INTERFACE I_Table EXTENDS __System.IQueryInterface

PROPERTY INTERNAL _InternalTable : REFERENCE TO ST_NciFeedGroupTable
GET
END_GET
END_PROPERTY

METHOD AddAxisDynamics : BOOL
VAR_INPUT
	displayIndex : UDINT;
    axis : I_Axis;
    acceleration : LREAL(0.000001-99999999);
    deceleration : LREAL(0.000001-99999999);
    jerk: LREAL(0.000001-99999999);
END_VAR
END_METHOD

METHOD AddBaseFrame : BOOL
VAR_INPUT
    displayIndex : UDINT;
    shiftX : LREAL;
    shiftY : LREAL;
    shiftZ : LREAL;
    rotationX : LREAL;
    rotationY : LREAL;
    rotationZ : LREAL;
    shiftQ1 : LREAL;
    shiftQ2 : LREAL;
    shiftQ3 : LREAL;
    shiftQ4 : LREAL;
    shiftQ5 : LREAL;
END_VAR
END_METHOD

METHOD AddBaseFrame3D : BOOL
VAR_INPUT
    displayIndex : UDINT;
    shiftX : LREAL;
    shiftY : LREAL;
    shiftZ : LREAL;
    rotationX : LREAL;
    rotationY : LREAL;
    rotationZ : LREAL;
END_VAR
END_METHOD

METHOD AddBezier3rdOrder : BOOL
VAR_INPUT
	displayIndex : UDINT;
    controlPoint1X : LREAL;
    controlPoint1Y : LREAL;
    controlPoint1Z : LREAL;
    controlPoint2X : LREAL;
    controlPoint2Y : LREAL;
    controlPoint2Z : LREAL;
	endPositionX : LREAL;
	endPositionY : LREAL;
	endPositionZ : LREAL;
	endPositionQ1 : LREAL;
	endPositionQ2 : LREAL;
	endPositionQ3 : LREAL;
	endPositionQ4 : LREAL;
	endPositionQ5 : LREAL;
	velocity : LREAL(0.000001-99999999);
	accurateStop : BOOL; // velocity at end == 0
END_VAR
END_METHOD

METHOD AddBezier3rdOrder3D : BOOL
VAR_INPUT
	displayIndex : UDINT;
    controlPoint1X : LREAL;
    controlPoint1Y : LREAL;
    controlPoint1Z : LREAL;
    controlPoint2X : LREAL;
    controlPoint2Y : LREAL;
    controlPoint2Z : LREAL;
	endPositionX : LREAL;
	endPositionY : LREAL;
	endPositionZ : LREAL;
	velocity : LREAL(0.000001-99999999);
	accurateStop : BOOL; // velocity at end == 0
END_VAR
END_METHOD

METHOD AddBezier5thOrder : BOOL
VAR_INPUT
	displayIndex : UDINT;
    controlPoint1X : LREAL;
    controlPoint1Y : LREAL;
    controlPoint1Z : LREAL;
    controlPoint2X : LREAL;
    controlPoint2Y : LREAL;
    controlPoint2Z : LREAL;
    controlPoint3X : LREAL;
    controlPoint3Y : LREAL;
    controlPoint3Z : LREAL;
    controlPoint4X : LREAL;
    controlPoint4Y : LREAL;
    controlPoint4Z : LREAL;
	endPositionX : LREAL;
	endPositionY : LREAL;
	endPositionZ : LREAL;
	endPositionQ1 : LREAL;
	endPositionQ2 : LREAL;
	endPositionQ3 : LREAL;
	endPositionQ4 : LREAL;
	endPositionQ5 : LREAL;
	velocity : LREAL(0.000001-99999999);
	accurateStop : BOOL; // velocity at end == 0
END_VAR
END_METHOD

METHOD AddBezier5thOrder3D : BOOL
VAR_INPUT
	displayIndex : UDINT;
    controlPoint1X : LREAL;
    controlPoint1Y : LREAL;
    controlPoint1Z : LREAL;
    controlPoint2X : LREAL;
    controlPoint2Y : LREAL;
    controlPoint2Z : LREAL;
    controlPoint3X : LREAL;
    controlPoint3Y : LREAL;
    controlPoint3Z : LREAL;
    controlPoint4X : LREAL;
    controlPoint4Y : LREAL;
    controlPoint4Z : LREAL;
	endPositionX : LREAL;
	endPositionY : LREAL;
	endPositionZ : LREAL;
	velocity : LREAL(0.000001-99999999);
	accurateStop : BOOL; // velocity at end == 0
END_VAR
END_METHOD

METHOD AddCircleCIP : BOOL
VAR_INPUT
	displayIndex : UDINT;
	endPositionX : LREAL;
	endPositionY : LREAL;
	endPositionZ : LREAL;
	arcPointX : LREAL;
	arcPointY : LREAL;
	arcPointZ : LREAL;
	endPositionQ1 : LREAL;
	endPositionQ2 : LREAL;
	endPositionQ3 : LREAL;
	endPositionQ4 : LREAL;
	endPositionQ5 : LREAL;
	velocity : LREAL(0.000001-99999999);
	accurateStop : BOOL; // velocity at end == 0
END_VAR
END_METHOD

METHOD AddCircleCIP3D : BOOL
VAR_INPUT
	displayIndex : UDINT;
	endPositionX : LREAL;
	endPositionY : LREAL;
	endPositionZ : LREAL;
	arcPointX : LREAL;
	arcPointY : LREAL;
	arcPointZ : LREAL;
	velocity : LREAL(0.000001-99999999);
	accurateStop : BOOL; // velocity at end == 0
END_VAR
END_METHOD

METHOD AddCircleOnPlane : BOOL
VAR_INPUT
	displayIndex : UDINT;
	endPositionX : LREAL;
	endPositionY : LREAL;
	endPositionZ : LREAL;
	centerX : LREAL;
	centerY : LREAL;
	centerZ : LREAL;
	endPositionQ1 : LREAL;
	endPositionQ2 : LREAL;
	endPositionQ3 : LREAL;
	endPositionQ4 : LREAL;
	endPositionQ5 : LREAL;
	plane : StandardPlane := StandardPlane.XY;
	clockwise : BOOL;
	velocity : LREAL(0.000001-99999999);
	accurateStop : BOOL; // velocity at end == 0
END_VAR
END_METHOD

METHOD AddCircleOnPlane3D : BOOL
VAR_INPUT
	displayIndex : UDINT;
	endPositionX : LREAL;
	endPositionY : LREAL;
	endPositionZ : LREAL;
	centerX : LREAL;
	centerY : LREAL;
	centerZ : LREAL;
	plane : StandardPlane := StandardPlane.XY;
	clockwise : BOOL;
	velocity : LREAL(0.000001-99999999);
	accurateStop : BOOL; // velocity at end == 0
END_VAR
END_METHOD

METHOD AddDwellTime : BOOL
VAR_INPUT
	displayIndex : UDINT;
    dwellTime : LREAL(0.000001-99999999); // seconds
END_VAR
END_METHOD

METHOD AddFeedrateInterpolation : BOOL
VAR_INPUT
	displayIndex : UDINT;
	interpolationType : FeedrateInterpolation;
END_VAR
END_METHOD

METHOD AddLine : BOOL
VAR_INPUT
    displayIndex: UDINT;
    endPositionX: LREAL;
    endPositionY: LREAL;
    endPositionZ: LREAL;
    endPositionQ1: LREAL;
    endPositionQ2: LREAL;
    endPositionQ3: LREAL;
    endPositionQ4: LREAL;
    endPositionQ5: LREAL;
    velocity: LREAL(0.000001-99999999);
    rapidTraverse: BOOL;
    accurateStop: BOOL; // velocity at end == 0
END_VAR
END_METHOD

METHOD AddLine3D : BOOL
VAR_INPUT
    displayIndex: UDINT;
    endPositionX: LREAL;
    endPositionY: LREAL;
    endPositionZ: LREAL;
    velocity: LREAL(0.000001-99999999);
    rapidTraverse: BOOL;
    accurateStop: BOOL; // velocity at end == 0
END_VAR
END_METHOD

METHOD AddMFunctionWithHandshake : BOOL
VAR_INPUT
	displayIndex : UDINT;
    functionNumber : INT(0..159);
END_VAR
END_METHOD

METHOD AddPathDynamics : BOOL
VAR_INPUT
    displayIndex : UDINT;
    acceleration : LREAL(0.000001-99999999);
    deceleration : LREAL(0.000001-99999999);
    jerk : LREAL(0.000001-99999999);
END_VAR
END_METHOD

METHOD AddStart : BOOL
VAR_INPUT
	x : LREAL;
	y : LREAL;
	z : LREAL;
	q1 : LREAL;
	q2 : LREAL;
	q3 : LREAL;
	q4 : LREAL;
	q5 : LREAL;
END_VAR
END_METHOD

METHOD AddStart3D : BOOL
VAR_INPUT
	x : LREAL;
	y : LREAL;
	z : LREAL;
END_VAR
END_METHOD

METHOD DisableTangentialFollowing : BOOL
END_METHOD

METHOD DisableVertexSmoothing : BOOL
VAR_INPUT
	displayIndex : UDINT;
END_VAR
END_METHOD

METHOD EnableTangentialFollowing : BOOL
VAR_INPUT
    tangentialAxis : NciAxis; // axis used for tangential following
    pathAxis1 : NciAxis; // describing the plane e.g. x
    pathAxis2 : NciAxis; // e.g. y ==> g17, xy plane
    offset : LREAL; // geo tangent is 0 degree, counting is mathmatical positive
	criticalAngle : LREAL(0.000001-90);
    behaviour : TangentialFollowingBehaviour;
END_VAR
END_METHOD

METHOD EnableVertexSmoothing : BOOL
VAR_INPUT
	displayIndex : UDINT;
	blendType : VertexSmoothingBlendingType;
	subType : VertexSmoothingSubType; 
	radius : LREAL(0.000001-99999999);
END_VAR
END_METHOD

METHOD End : BOOL
END_METHOD

PROPERTY ErrorId : UDINT
GET
END_GET
END_PROPERTY

PROPERTY FilledRows : INT
GET
END_GET
END_PROPERTY

PROPERTY HasError : BOOL
GET
END_GET
END_PROPERTY

METHOD ResetAll : BOOL
END_METHOD

METHOD ResetTable : BOOL
END_METHOD

END_INTERFACE

(* stored: Version 1.1.0.1, ProductVersion 3.1.4024.12
   Itf I_Table: Id {739dd892-cb31-4bd0-a191-42ac4941c726}
   Property _InternalTable: Id {7b598730-f029-415a-b056-55b65e711f78}
   Get Get: Id {078af100-b2d1-44ec-a028-70c3bd4f11fe}
   Method AddAxisDynamics: Id {90b05305-7afb-4b84-85bb-ee24976dbbd8}
   Method AddBaseFrame: Id {afffafb0-7905-4a68-8a9d-9d617c15ab24}
   Method AddBaseFrame3D: Id {f4614335-b82a-47c3-9bee-2b6d18723083}
   Method AddBezier3rdOrder: Id {dac5ed2d-a91b-48eb-9950-3b9fb425d0a0}
   Method AddBezier3rdOrder3D: Id {4da67f00-46f0-416b-99fe-34dfe230497f}
   Method AddBezier5thOrder: Id {608ada7a-5786-4b63-adf2-4f2f4d22b371}
   Method AddBezier5thOrder3D: Id {5448bb54-6ec0-455c-b5b5-abe54411ded6}
   Method AddCircleCIP: Id {f044aea4-54b1-4049-a247-70896b69338f}
   Method AddCircleCIP3D: Id {326bb761-f8b9-428d-b787-7723655c4754}
   Method AddCircleOnPlane: Id {b4aaee45-5a64-4c78-bb6f-16a1f9e654e4}
   Method AddCircleOnPlane3D: Id {c9bf8cb5-0c5c-4f90-b503-fe16026c8d3f}
   Method AddDwellTime: Id {b6adeded-8b48-4167-8093-b8d002dcc967}
   Method AddFeedrateInterpolation: Id {5d6f284c-2f7d-4fbf-b57d-9c01ad6226bb}
   Method AddLine: Id {106e0278-8d7e-41d7-b6ef-895917ab3f3a}
   Method AddLine3D: Id {99855279-ecd0-41f0-99b1-2a5b21a9a526}
   Method AddMFunctionWithHandshake: Id {5f20215b-a091-4387-af2a-b5cdbe2e7b1b}
   Method AddPathDynamics: Id {3d54cbd2-cb38-43da-a49d-c93565722659}
   Method AddStart: Id {f3b32d87-ed5b-4ff7-ab74-18ab3d304a5b}
   Method AddStart3D: Id {1ee68d1d-485d-4f29-b4d1-78f0bd4ad3fa}
   Method DisableTangentialFollowing: Id {b0c3e73a-02de-4535-a428-d2afc05f3630}
   Method DisableVertexSmoothing: Id {e2c24514-b215-47a0-ab5e-791ad29a1996}
   Method EnableTangentialFollowing: Id {d1542920-828f-4dc4-bb27-e38798603e0a}
   Method EnableVertexSmoothing: Id {4a6ad671-c0c0-409a-bd30-08442afd78af}
   Method End: Id {83e2a824-c91c-4b2c-be28-ca32c6009d21}
   Property ErrorId: Id {88f45720-8df7-4ae7-a4d0-027d75f3ccab}
   Get Get: Id {d03d66d0-6f0d-4d47-9e45-05d01b43b308}
   Property FilledRows: Id {4da66c5b-4512-4aed-9d63-8e9759611ae8}
   Get Get: Id {3817b9df-e215-4c87-b43d-10c299f003c8}
   Property HasError: Id {bc358fad-d2e1-4362-9d3a-cf1385ec4e86}
   Get Get: Id {218b2313-e6f5-4eeb-ae3b-e776fbba6cd5}
   Method ResetAll: Id {f8ec2ce9-b498-4d27-8681-547ca524a446}
   Method ResetTable: Id {57ebc5eb-e485-43b2-a962-0a43a9dff7df} *)
